{attribute 'linkalways'}
{attribute 'hide_all_locals'}
FUNCTION_BLOCK ValueUintRead EXTENDS ValueBase IMPLEMENTS ValueRead
VAR
	thisValue : UINT;
END_VAR

{attribute 'call_after_global_init_slot' := '1'}
{attribute 'call_after_online_change_slot' := '1'}
METHOD PROTECTED GetThisAnyType
VAR_INPUT
END_VAR
thisAnyType := ToAnyType(thisValue);
END_METHOD

METHOD GetAsType : BOOL
VAR_INPUT
	destination : __SYSTEM.AnyType;
END_VAR
GetAsType := ConvertAnyType(thisAnyType, destination);
END_METHOD

METHOD GetAsString : T_MaxString
VAR_INPUT
END_VAR
GetAsString := TO_STRING(thisValue);
END_METHOD

METHOD Get : BOOL
VAR_INPUT
	destination : ANY;
END_VAR
Get := ConvertAnyType(thisAnyType, destination);
END_METHOD

METHOD FB_init : BOOL
VAR_INPUT
	bInitRetains : BOOL; // if TRUE, the retain variables are initialized (warm start / cold start)
	bInCopyCode : BOOL;  // if TRUE, the instance afterwards gets moved into the copy code (online change)
END_VAR
_ValueType := __SYSTEM.TYPE_CLASS.TYPE_UINT;
END_METHOD

{attribute 'monitoring' := 'call'}
PROPERTY Value : UINT
GET
Value := thisValue;
END_GET
END_PROPERTY

END_FUNCTION_BLOCK

(* stored: Version 1.1.0.1
   POU ValueUintRead: Id {a93c3131-5582-43f2-9f10-9246147157b2}, SpecialFunc None
   Method GetThisAnyType: Id {612ed96d-c948-4461-ade8-b91c21312b20}
   Method GetAsType: Id {ca5293e5-c605-45d3-af0a-30c7fc69dc01}
   Method GetAsString: Id {df457ac2-aea0-4fa7-b51e-1b091bda1242}
   Method Get: Id {8ad85e45-adbe-43b8-89b8-671c53a39319}
   Method FB_init: Id {fb9c68de-55cb-4725-bac2-e0d23aba2d2a}
   Property Value: Id {8341b9a2-65ad-4fdc-9f3e-8fd1c4b16fc0}
   Get Get: Id {c604bfae-afd2-4f3e-b3fb-164494ddd4ec} *)
